(* PLC project Tc2_IoFunctions.IOF_GetDeviceIDByName Demo, tc3-libraries-kb TwinCAT 3.1 *)
(* stored: creationDateTime 2026-05-21T00:00:00, modificationDateTime 2026-05-21T00:00:00 *)

PROGRAM P_Demo_IOF_GetDeviceIDByName
  VAR
    fbLookupDeviceId : IOF_GetDeviceIDByName;  (* 设备名 → ID FB *)
    sTargetNetId : T_AmsNetId := '';  (* 本机 *)
    sLookupDeviceName : T_MaxString := 'DP_Master_Main';  (* 设备名字（区分大小写） *)
    bStartLookupDeviceId : BOOL := FALSE;  (* 上升沿触发 *)
    tLookupTimeout : TIME := T#5S;  (* 超时 *)
    bLookupBusy : BOOL;  (* 工作中 *)
    bLookupError : BOOL;  (* 失败 *)
    nLastErrCode : UDINT;  (* 错误号 *)
    nLookedUpDeviceId : UDINT;  (* 查得 Device Id *)
  END_VAR

// =============================================================================
// 场景：程序需要按设备名字定位 Profibus 主站做后续操作，避免硬编码 ID。
// 价值：与工程配置同步：改 ID 不影响 PLC 程序，只要名字不改。
// 验证：登录后 sLookupDeviceName := "DP_Master_Main"，在线写 bStartLookupDeviceId := TRUE → 回 FALSE 后 nLookedUpDeviceId 显示 System Manager 中分配给该设备的 Device Id。
// 验证步骤：
//   1. 右键 PLC 项目 → Import PLCopenXML → 选本文件
//   2. 引用 Tc2_IoFunctions（References → Add library）
//   3. 编译 → 登录 → 运行；按上方『验证』行的指示在线写值观察
// =============================================================================

fbLookupDeviceId(
    NETID      := sTargetNetId,
    DEVICENAME := sLookupDeviceName,
    START      := bStartLookupDeviceId,
    TMOUT      := tLookupTimeout,
    BUSY       => bLookupBusy,
    ERR        => bLookupError,
    ERRID      => nLastErrCode,
    DEVICEID   => nLookedUpDeviceId
);
END_PROGRAM
